{attribute 'GeneratedUsingTerminal: EL6861-0000-0016'}
{attribute addProperty BoxType "EL6861-0000-0016"}
{attribute addProperty Id "EtcSlaveTerminalBaseCOM_TxPDO_Map_InputsAT %I*COM_TxPDO_Map_Inputs_93BAD1D7137COM_RxPDO_MapAT %Q*COM_RxPDO_Map_01DE24DC133WcStateAT %I*WcState_9091E0EB2InfoDataAT %I*InfoData_32EB74EA10"}
{attribute addProperty CRC "3553568871"}
{attribute addProperty Size "282"}
TYPE EL6861_D3CF2867 EXTENDS EtcSlaveTerminalBase :
STRUCT
	{attribute addProperty Name "COM_TxPDO_Map_Inputs"}
	COM_TxPDO_Map_Inputs : COM_TxPDO_Map_Inputs_93BAD1D7;
	{attribute addProperty Name "COM_RxPDO_Map"}
	COM_RxPDO_Map : COM_RxPDO_Map_01DE24DC;
	{attribute addProperty Name "WcState"}
	WcState : WcState_9091E0EB;
	{attribute addProperty Name "InfoData"}
	InfoData : InfoData_32EB74EA;
END_STRUCT
END_TYPE

(* stored: Version 1.2.0.0, ProductVersion 3.1.4024.9
   DUT EL6861_D3CF2867: Id {ce4eb60c-ab68-40aa-8c6f-4e350863d540} *)
